Fanuc KAREL source: kb00016.KL

-- PROVISIONAL review KL for V1013-1; original PC SHA256 cc7e058f570604768854e5abac9d17518ff4fdc89d49111cb3d7394d68ccdc2c
-- Incomplete behavior may be omitted. Consult companion uncertainty JSON. Do not deploy.
PROGRAM KB00016
%NOLOCKGROUP
BEGIN
  -- UNRESOLVED_PC offsets 5-14; opcodes 3F,75
  -- UNRESOLVED_PC offsets 19-26; opcodes 9D,23
  -- UNRESOLVED_PC offsets 31-38; opcodes 9D,23
  -- UNRESOLVED_PC offsets 43-50; opcodes 9D,23
  -- UNRESOLVED_PC offsets 55-85; opcodes 27,22,2A,22,22,22,31
  -- UNRESOLVED_PC offsets 90-94; opcodes 7F
END KB00016
